{attribute 'GeneratedUsingTerminal: EL3413-0000-0016'}
{attribute addProperty BoxType "EL3413-0000-0016"}
{attribute addProperty Id "TxPDO_ToggleBOOL1"}
{attribute addProperty CRC "1378780365"}
{attribute addProperty Size "1"}
TYPE STATUS_522E84CD :
STRUCT
	{attribute addProperty Name "TxPDO_Toggle"}
	TxPDO_Toggle : BOOL;
END_STRUCT
END_TYPE

(* stored: Version 1.2.0.0, ProductVersion 3.1.4024.9
   DUT STATUS_522E84CD: Id {13b70bc2-f4e4-466a-ba43-67788ea906a4} *)
